FUNCTION_BLOCK PUBLIC ElmoVelocityCtrlAxis_FB EXTENDS VelocityCtrlAxis_FB  
VAR_INPUT
	

END_VAR

VAR_OUTPUT
END_VAR
	
VAR

	
END_VAR

SUPER^();

METHOD METH_ChangeToVelMode : BOOL
VAR_INPUT
	Execute : BOOL;
END_VAR
IF InitSctrlTrigger.EDGEPOS( Execute) THEN
	CngToVelocityState := 1;
	METH_ChangeToVelMode := FALSE;
	rAxisBasicFB.AxisCtrlPtr^.Input.Command.Power := FALSE;
	
	OldCyclicTorque := 0;		
	OldSctrlKp 		:= 0;
	OldSctrlKi 		:= 0;			
	rAxisBasicFB.Meth_WriteObj (FALSE, enumMotionobject.OPERATION_MODE, TO_LREAL(eDriveModeOfOperation.CyclicSyncVelocity));

END_IF

IF InitSctrlTrigger.EDGENEG( Execute) THEN
	CngToVelocityState := 0;
END_IF


CASE CngToVelocityState OF
	0:
		METH_ChangeToVelMode := FALSE;
	1:
		IF ReadPosCtrlParamDone = FALSE THEN
			 Meth_ReadPosCtrlValues(FALSE);
			 CngToVelocityState := CngToVelocityState +1;	
		ELSE
			CngToVelocityState := CngToVelocityState +2;
		END_IF		
	2:
		IF Meth_ReadPosCtrlValues(TRUE) THEN
			
			rAxisBasicFB.Meth_WriteObj (FALSE, enumMotionobject.OPERATION_MODE,eDriveModeOfOperation.CyclicSyncVelocity);
			
			CngToVelocityState := CngToVelocityState +1;
			
		END_IF
	3:	//Change mode to velocity control
		IF rAxisBasicFB.Meth_WriteObj (TRUE, enumMotionobject.OPERATION_MODE,eDriveModeOfOperation.CyclicSyncVelocity) THEN			
			rAxisBasicFB.Meth_WriteObj (FALSE, enumMotionobject.OPERATION_MODE,eDriveModeOfOperation.CyclicSyncVelocity);
			CngToVelocityState := CngToVelocityState +1;
		END_IF
		
	4://Disable Gain Control
		IF NOT rAxisBasicFB.AxisCtrlPtr^.Output.Status.MC_Power.Status THEN
			IF rAxisBasicFB.Meth_WriteObj (TRUE, enumMotionobject.GAIN_SCHEDULE,0) THEN			
				rAxisBasicFB.Meth_WriteObj (FALSE, enumMotionobject.OPERATION_MODE,eDriveModeOfOperation.CyclicSyncVelocity);			
				CngToVelocityState := CngToVelocityState +1;
			END_IF
		END_IF	
	
	5:	
		rAxisBasicFB.AxisCtrlPtr^.Input.Command.Power := TRUE;
		IF rAxisBasicFB.AxisCtrlPtr^.Output.Status.AxisStatus.StandStill THEN
			CngToVelocityState := CngToVelocityState +1;
		END_IF
	6:
		IF  rAxisBasicFB.Meth_WriteObj(TRUE, enumMotionObject.ACC_CLOSE_POS_ERR ,   rVelocityCtrl.Input.Parameter.CyclicVelocity    , Error =>Error ) THEN
			rAxisBasicFB.Meth_WriteObj(FALSE, enumMotionObject.ACC_CLOSE_POS_ERR ,0 );
			CngToVelocityState := CngToVelocityState +1;
		END_IF	
	
	7:	
		METH_ChangeToVelMode := TRUE;
END_CASE
END_METHOD

METHOD Meth_InitSctrl : BOOL
VAR_INPUT
	Execute : BOOL;
END_VAR


VAR_OUTPUT
	Error : BOOL;
END_VAR
IF InitSctrlTrigger.EDGEPOS(Execute) THEN
	InitSctrlState  := 1;
	Meth_InitSctrl := FALSE;
	rAxisBasicFB.Meth_InitVelKP (FALSE,0);
	rAxisBasicFB.Meth_InitVelKI(FALSE,0);
	Error := FALSE;
END_IF


IF InitSctrlTrigger.EDGENEG(Execute) THEN
	
	 InitSctrlState:= 0;
END_IF


CASE InitSctrlState OF
 
		
	1:
		 			
	 
	 	IF rAxisBasicFB.Meth_InitVelKP (TRUE,(rVelocityCtrl.Input.Parameter.SctrlKp), Error=>Error) THEN
	 		OldSctrlKp := rVelocityCtrl.Input.Parameter.SctrlKp;
	 		InitSctrlState := InitSctrlState +1;
	 		rAxisBasicFB.Meth_InitVelKP (FALSE,rVelocityCtrl.Input.Parameter.SctrlKp);
	 	END_IF	
 	  
			

	2:
	
			IF rAxisBasicFB.Meth_InitVelKI(TRUE,(rVelocityCtrl.Input.Parameter.SctrlKi), Error=>Error) THEN
				rAxisBasicFB.Meth_InitVelKP (FALSE,rVelocityCtrl.Input.Parameter.SctrlKi);
				OldSctrlKi := rVelocityCtrl.Input.Parameter.SctrlKi ;
				InitSctrlState := InitSctrlState +1;
			END_IF	

		IF Error THEN
		//	
		END_IF
		
	3:		
		rVelocityCtrl.Output.Status.SctrlInitialized := TRUE;
		Meth_InitSctrl := TRUE; 
	END_CASE
END_METHOD

METHOD Meth_ReadPosCtrlValues : BOOL
VAR_INPUT
	Execute : BOOL;
END_VAR


VAR_INST
	// Service Functions Variablea
	ReadPosCtrlTrigger : Trigger ;
	ReadPosCtrlState   : SINT;
END_VAR	

VAR_OUTPUT
	Error : BOOL;	
END_VAR
IF ReadPosCtrlTrigger.EDGEPOS(Execute) THEN
	ReadPosCtrlState  := 1;
	Meth_ReadPosCtrlValues := FALSE;
	Error := FALSE;
	rAxisBasicFB.Meth_ReadObj(FALSE, enumMotionObject.MAX_TORQUE, Value =>rVelocityCtrl.Output.monitor.OrgMaxTorque, Error =>Error );
END_IF


IF ReadPosCtrlTrigger.EDGENEG(Execute) THEN
	 rAxisBasicFB.Meth_ReadObj(FALSE, enumMotionObject.MAX_TORQUE, Value =>rVelocityCtrl.Output.monitor.OrgMaxTorque, Error =>Error );
	 ReadPosCtrlState:= 0;
END_IF


CASE ReadPosCtrlState OF
 
	1:
		IF  rAxisBasicFB.Meth_ReadObj(TRUE, enumMotionObject.TORQUE_OFFSET, Value =>rVelocityCtrl.Output.monitor.OrgCyclicTorque, Error =>Error ) THEN
			rAxisBasicFB.Meth_ReadObj(FALSE, enumMotionObject.TORQUE_OFFSET  );
 			ReadPosCtrlState := ReadPosCtrlState +1;
			Error := FALSE;						
		END_IF
		IF Error THEN
			ReadPosCtrlState := 33;
		END_IF
			
	2:
		IF  rAxisBasicFB.Meth_ReadObj(TRUE, enumMotionObject.VEL_KP, Value =>rVelocityCtrl.Output.monitor.OrgSctrlKp, Error =>Error ) THEN
			rVelocityCtrl.Output.monitor.OrgVelKp := rVelocityCtrl.Output.monitor.OrgSctrlKp;
			rAxisBasicFB.Meth_ReadObj(FALSE, enumMotionObject.TORQUE_OFFSET  );
 			ReadPosCtrlState := ReadPosCtrlState +1;
		END_IF
	3:
		IF  rAxisBasicFB.Meth_ReadObj(TRUE, enumMotionObject.VEL_KI, Value =>rVelocityCtrl.Output.monitor.OrgSctrlKi, Error =>Error ) THEN
			rAxisBasicFB.Meth_ReadObj(FALSE, enumMotionObject.TORQUE_OFFSET  );
 			ReadPosCtrlState := ReadPosCtrlState +1;
		END_IF
	
	4:
		IF rAxisBasicFB.Meth_ReadObj (TRUE, enumMotionobject.GAIN_SCHEDULE, Value =>rVelocityCtrl.Output.monitor.OrgGainCtrl, Error =>Error) THEN			
				rAxisBasicFB.Meth_ReadObj(FALSE, enumMotionObject.TORQUE_OFFSET  );
				ReadPosCtrlState := ReadPosCtrlState +1;						
		END_IF		
		
	5:
			IF rAxisBasicFB.Meth_ReadObj (TRUE, enumMotionobject.ACC_CLOSE_POS_ERR, Value =>rVelocityCtrl.Output.monitor.OrgAccToCloseThePosError, Error =>Error) THEN			
				rAxisBasicFB.Meth_ReadObj(FALSE, enumMotionObject.TORQUE_OFFSET  );
				ReadPosCtrlState := ReadPosCtrlState +1;						
			END_IF	
	6:	
		IF rAxisBasicFB.Meth_ReadObj (TRUE, enumMotionobject.MAX_TORQUE  , Value =>rVelocityCtrl.Output.monitor.OrgMaxTorque, Error =>Error) THEN	
				fnLogMsg(ADR(LogMsg_0),LOG_INFO,'MAX_TORQUE org=%d',TO_DINT(rVelocityCtrl.Output.monitor.OrgMaxTorque),0,0);		
				rAxisBasicFB.Meth_ReadObj(FALSE, enumMotionObject.TORQUE_OFFSET  );
				ReadPosCtrlState := ReadPosCtrlState +1;						
		 	END_IF		

	7:
	
				
		ReadPosCtrlParamDone := TRUE;
		Meth_ReadPosCtrlValues := TRUE; 
	END_CASE
END_METHOD

METHOD Meth_ReturnOrgPosCtrlValues : BOOL
VAR_INPUT
	Execute : BOOL;
END_VAR


VAR_INST
		// Service Functions Variablea
	ReturnOrgTrigger : Trigger ;
	ReturnOrgState   : SINT;
END_VAR	

VAR_OUTPUT
	Error : BOOL;
END_VAR
IF ReturnOrgTrigger.EDGEPOS(Execute) THEN
	ReturnOrgState  := 1;
	Meth_ReturnOrgPosCtrlValues := FALSE;
	Error := FALSE;
	rAxisBasicFB.Meth_WriteObj(FALSE, enumMotionObject.MAX_TORQUE, rVelocityCtrl.Output.monitor.OrgMaxTorque, Error =>Error );
END_IF


IF ReturnOrgTrigger.EDGENEG(Execute) THEN
	 rAxisBasicFB.Meth_WriteObj(FALSE, enumMotionObject.MAX_TORQUE,  rVelocityCtrl.Output.monitor.OrgMaxTorque, Error =>Error );
	 ReturnOrgState:= 0;
END_IF


CASE ReturnOrgState OF
 
		
	1:	
		IF  rAxisBasicFB.Meth_WriteObj(TRUE, enumMotionObject.GAIN_SCHEDULE,  rVelocityCtrl.Output.monitor.OrgGainCtrl, Error =>Error ) THEN
			rAxisBasicFB.Meth_WriteObj(FALSE, enumMotionObject.GAIN_SCHEDULE ,0 );
 			ReturnOrgState := ReturnOrgState +1;
		END_IF		
			
	2:
		IF  rAxisBasicFB.Meth_WriteObj(TRUE, enumMotionObject.VEL_KP,  rVelocityCtrl.Output.monitor.OrgSctrlKp, Error =>Error ) THEN
			rAxisBasicFB.Meth_WriteObj(FALSE,enumMotionObject.VEL_KP,0  );
 			ReturnOrgState := ReturnOrgState +1;
		END_IF
	3:
		IF  rAxisBasicFB.Meth_WriteObj(TRUE, enumMotionObject.VEL_KI,  rVelocityCtrl.Output.monitor.OrgSctrlKi, Error =>Error ) THEN
			rAxisBasicFB.Meth_WriteObj(FALSE, enumMotionObject.VEL_KP ,0 );
 			ReturnOrgState := ReturnOrgState +1;
		END_IF
	
	4:
		IF  rAxisBasicFB.Meth_WriteObj(TRUE, enumMotionObject.TORQUE_OFFSET, rVelocityCtrl.Output.monitor.OrgCyclicTorque , Error =>Error ) THEN
			rAxisBasicFB.Meth_WriteObj(FALSE, enumMotionObject.VEL_KP ,0 );
 			ReturnOrgState := ReturnOrgState +1;
		END_IF
		
	5:				
		IF  rAxisBasicFB.Meth_WriteObj(TRUE, enumMotionObject.MAX_TORQUE, rVelocityCtrl.Output.monitor.OrgMaxTorque  , Error =>Error ) THEN
			rAxisBasicFB.Meth_WriteObj(FALSE, enumMotionObject.VEL_KP ,0 );
 			ReturnOrgState := ReturnOrgState +1;
		END_IF
	6:	
		ReadPosCtrlParamDone := TRUE;
		Meth_ReturnOrgPosCtrlValues := TRUE; 
	END_CASE
END_METHOD

END_FUNCTION_BLOCK

(* stored: Version 1.1.0.1, ProductVersion 3.1.4024.3
   POU ElmoVelocityCtrlAxis_FB: Id {32652808-323a-4d40-8e6e-e6eb3fbe0c89}, SpecialFunc None
   Method METH_ChangeToVelMode: Id {c9646577-c354-412a-b857-49145aeed4a6}
   Method Meth_InitSctrl: Id {48a91f68-467f-4b94-9de6-7ca1cc0c4e6b}
   Method Meth_ReadPosCtrlValues: Id {8ed33566-9eb0-445e-b8b4-88f1340b1182}
   Method Meth_ReturnOrgPosCtrlValues: Id {8c8cd9c8-8bc8-4d0e-88cc-047c112dcad3} *)
